{region '#Template'}
	{attribute 'Category' := 'Universal'}
	{attribute 'Version' := '0.0.1.0'}
	{attribute 'Tags' := 'Universal, Pump'}
	{attribute 'Description' := 'Pumpe 1 stufig	// Pump 1 stage'}
{endregion}
FUNCTION_BLOCK FB_BA_Pu1st EXTENDS FB_BA_Mot1st
VAR_INPUT
	bAblkLock				: BOOL;	
END_VAR
VAR_INPUT CONSTANT
	DlyOff					: FB_BA_DlyOff;								
	Ablk					: FB_BA_AntiBlocking;							
END_VAR
VAR
	PrioSwiPgm				: FB_BA_PrioSwi_B04;
END_VAR

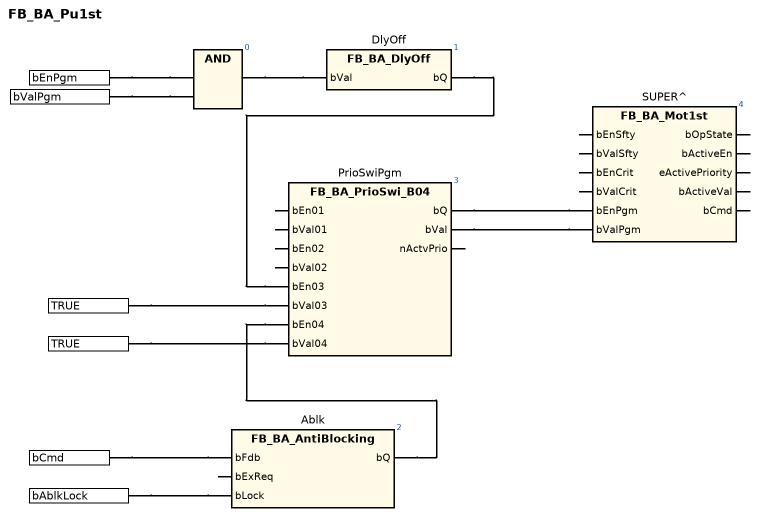
DlyOff(bVal := bEnPgm AND bValPgm); // FB_BA_DlyOff
// parameter Ablk.sObjectName := '[Idx=01]'
Ablk(bFdb := bCmd, bLock := bAblkLock); // FB_BA_AntiBlocking
PrioSwiPgm(bEn03 := DlyOff.bQ, bVal03 := TRUE, bEn04 := Ablk.bQ, bVal04 := TRUE); // FB_BA_PrioSwi_B04
SUPER^(bEnPgm := PrioSwiPgm.bQ, bValPgm := PrioSwiPgm.bVal); // FB_BA_Mot1st

METHOD FB_init : BOOL
VAR_INPUT
	bInitRetains : BOOL; // if TRUE, the retain variables are initialized (warm start / cold start)
	bInCopyCode : BOOL;  // if TRUE, the instance afterwards gets moved into the copy code (online change)
END_VAR
DlyOff.iParent			:= THIS^;	
DlyOff.iLabel			:= LblUniFieldDevice.Pump_DlyOff;
DlyOff.sObjectName		:= '{Idx=01}';									
DlyOff.eDPADMode		:= E_BA_DPADMode.eIncludeDescription;

Ablk.iParent			:= THIS^;	
Ablk.iLabel				:= LblUniFieldDevice.Pump_Ablk;
Ablk.sObjectName		:= '{Idx=01}';																	
Ablk.eDPADMode			:= E_BA_DPADMode.eIncludeDescription;
END_METHOD

END_FUNCTION_BLOCK

(* stored: Version 1.1.0.1, ProductVersion 3.1.4024.6
   POU FB_BA_Pu1st: Id {53959648-a10b-4004-95a8-19d60da429e0}, SpecialFunc None
   Method FB_init: Id {8ab03f2e-99d0-40d4-ae99-798d8cb41cef} *)
